FUNCTION_BLOCK GEN_PULSE_DIST (* Distance based Impulse Generator *)
  (* Standard: 61499-1; Description: Distance based Impulse Generator START with a HIGH Pulse. *)
  (* Version 1.0, 2024-10-18, franz *)
  PACKAGE signalprocessing_plus::distance;
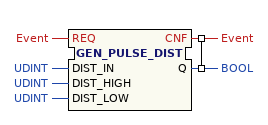
  EVENT_INPUT
    REQ; (* Normal Execution Request *)
  END_EVENT
  EVENT_OUTPUT
    CNF WITH Q; (* Execution Confirmation *)
  END_EVENT
  VAR_INPUT
    DIST_IN : UDINT; (* Travelled Distance *)
    DIST_HIGH : UDINT; (* Distance for Output HIGH *)
    DIST_LOW : UDINT; (* Distance for Output LOW *)
  END_VAR
  VAR_OUTPUT
    Q : BOOL; (* Output *)
  END_VAR
  VAR
    DIST_REMAINDER : UDINT;
  END_VAR
  ALGORITHM REQ IN ST:
DIST_REMAINDER := DIST_IN MOD (DIST_HIGH + DIST_LOW);

IF (DIST_REMAINDER >= DIST_HIGH) THEN
	Q := TRUE;
ELSE
	Q := FALSE;
END_IF;
  END_ALGORITHM
END_FUNCTION_BLOCK
